{attribute 'qualified_only'}
{attribute 'strict'}
TYPE E_STREAMSEEKTYPE :
(
	Origin := 0,
	Current,
	Current_Reversed,
	End
);
END_TYPE

(* stored: Version 1.1.0.1, ProductVersion 3.1.4022.3
   DUT E_STREAMSEEKTYPE: Id {9dcce5c6-f8f2-479f-94ee-16435a85a014} *)
